// TIA Portal V16 export
// export: Created 2021-11-12T13:31:05.7445128Z, ExportSetting WithDefaults, DisplayName Totally Integrated Automation Portal, DisplayVersion V16 Update 3, DisplayName TIA Portal Version Control Interface, DisplayVersion V16 Update 2, DisplayName TIA Portal Openness, DisplayVersion V16 Update 3, DisplayName SINAMICS Startdrive Advanced, DisplayVersion V16 Update 5, DisplayName SINAMICS Startdrive G130, G150, S120, S150, SINAMICS MV, S210, DisplayVersion V16 Update 5, DisplayName SINAMICS Startdrive G110M, G120, G120C, G120D, G120P, G115D, DisplayVersion V16 Update 5, DisplayName STEP 7 Professional, DisplayVersion V16 Update 3, DisplayName STEP 7 Safety, DisplayVersion V16, DisplayName WinCC UA Professional, DisplayVersion V16 Update 3
DATA_BLOCK "Communication"   // DB12
{ S7_Optimized_Access := 'TRUE'; DB_Accessible_From_OPC_UA := 'FALSE' }
VERSION : 0.1
// stored: AutoNumber true, DBAccessibleFromOPCUA false, IsOnlyStoredInLoadMemory false, IsRetainMemResEnabled false, IsWriteProtectedInAS false, MemoryReserve 100
   VAR
      KAS1 : Struct   // Comunication saw KASTO 1
         IN : "UDT_COMM_KAS1_CRS";   // Inputs from saw KASTO1
         OUT : "UDT_COMM_CRS_KAS1";   // Outputs to saw KASTO1
      END_STRUCT;
      KAS2 : Struct   // Comunication saw KASTO 2
         IN : "UDT_COMM_KAS2_CRS";   // Inputs from saw KASTO2
         OUT : "UDT_COMM_CRS_KAS2";   // Outputs to saw KASTO2
      END_STRUCT;
      BSN1 : Struct   // Comunication owen BSN1
         IN : "UDT_COMM_BSN1_CRS";   // Inputs from owen BSN1
         OUT : "UDT_COMM_CRS_BSN1";   // Outputs to owen BSN1
      END_STRUCT;
      BSN2 : Struct   // Comunication owen BSN2
         IN : "UDT_COMM_BSN2_CRS";   // Inputs from owen BSN2
         OUT : "UDT_COMM_CRS_BSN2";   // Outputs to owen BSN2
      END_STRUCT;
      SCH1 : Struct   // Comunication press machine SCHULER1
         IN : "UDT_COMM_SCH1_CRS";   // Inputs from press machine SCHULER
         OUT : "UDT_COMM_CRS_SCH1";   // Outputs to press machine schuler
      END_STRUCT;
      BSN3 : Struct   // Comunication owen BSN3
         IN : "UDT_COMM_BSN3_CRS";   // Inputs from owen BSN3
         OUT : "UDT_COMM_CRS_BSN3";   // Outputs to owen BSN3
      END_STRUCT;
      BSN4 : Struct   // Comunication owen BSN4
         IN : "UDT_COMM_BSN4_CRS";   // Inputs from owen BSN4
         OUT : "UDT_COMM_CRS_BSN4";   // Outputs to owen BSN4
      END_STRUCT;
      BSN5 : Struct   // Comunication owen BSN5
         IN : "UDT_COMM_BSN5_CRS";   // Inputs from owen BSN5
         OUT : "UDT_COMM_CRS_BSN5";   // Outputs to owen BSN5
      END_STRUCT;
      THM1 : Struct   // Comunication blasting machine THROWAL1
         IN : "UDT_COMM_THM1_CRS";   // Inputs from blasting machine THROWAL1
         OUT : "UDT_COMM_CRS_THM1";   // Outputs to blasting machine THROWAL1
      END_STRUCT;
      THM2 : Struct   // Comunication blasting machine THROWAL2
         IN : "UDT_COMM_THM2_CRS";   // Inputs from blasting machine THROWAL2
         OUT : "UDT_COMM_CRS_THM2";   // Outputs to blasting machine THROWAL2
      END_STRUCT;
      MEM1 : Struct   // Comunication primary cooling system MEMTECH1
         IN : "UDT_COMM_MEM1_CRS";   // Inputs from cooling system MEMTECH
         OUT : "UDT_COMM_CRS_MEM1";   // Outputs to cooling system MEMTECH
      END_STRUCT;
   END_VAR
BEGIN
END_DATA_BLOCK
